FUNCTION_BLOCK FB_SXU
VAR_INPUT
	
END_VAR

VAR_OUTPUT
END_VAR



VAR
    // From lcls-srv01: grep -e KDes  /u1/lcls/epics/ioc/data/sioc-unds-uc*/iocInfo/IOC.pvlist |sort


    {attribute 'pytmc' := 'pv: 26; link: 2650:'}
    fbSegment_26 : FB_UndulatorSegment;
    
    {attribute 'pytmc' := 'pv: 27; link: 2750:'}
    fbSegment_27 : FB_UndulatorSegment;
    
    {attribute 'pytmc' := 'pv: 28; link: 2850:'}
    fbSegment_28 : FB_UndulatorSegment;
    
    {attribute 'pytmc' := 'pv: 29; link: 2950:'}
    fbSegment_29 : FB_UndulatorSegment;
    
    {attribute 'pytmc' := 'pv: 30; link: 3050:'}
    fbSegment_30 : FB_UndulatorSegment;
    
    {attribute 'pytmc' := 'pv: 31; link: 3150:'}
    fbSegment_31 : FB_UndulatorSegment;
    
    {attribute 'pytmc' := 'pv: 32; link: 3250:'}
    fbSegment_32 : FB_UndulatorSegment;
    
    {attribute 'pytmc' := 'pv: 33; link: 3350:'}
    fbSegment_33 : FB_UndulatorSegment;
    
    {attribute 'pytmc' := 'pv: 34; link: 3450:'}
    fbSegment_34 : FB_UndulatorSegment;
    
    {attribute 'pytmc' := 'pv: 36; link: 3650:'}
    fbSegment_36 : FB_UndulatorSegment;
    
    {attribute 'pytmc' := 'pv: 37; link: 3750:'}
    fbSegment_37 : FB_UndulatorSegment;
    
    {attribute 'pytmc' := 'pv: 38; link: 3850:'}
    fbSegment_38 : FB_UndulatorSegment;
    
    {attribute 'pytmc' := 'pv: 39; link: 3950:'}
    fbSegment_39 : FB_UndulatorSegment;
    
    {attribute 'pytmc' := 'pv: 40; link: 4050:'}
    fbSegment_40 : FB_UndulatorSegment;
    
    {attribute 'pytmc' := 'pv: 41; link: 4150:'}
    fbSegment_41 : FB_UndulatorSegment;
    
    {attribute 'pytmc' := 'pv: 42; link: 4250:'}
    fbSegment_42 : FB_UndulatorSegment;
    
    {attribute 'pytmc' := 'pv: 43; link: 4350:'}
    fbSegment_43 : FB_UndulatorSegment;
    
    {attribute 'pytmc' := 'pv: 44; link: 4450:'}
    fbSegment_44 : FB_UndulatorSegment;
    
    {attribute 'pytmc' := 'pv: 45; link: 4550:'}
    fbSegment_45 : FB_UndulatorSegment;
    
    {attribute 'pytmc' := 'pv: 46; link: 4650:'}
    fbSegment_46 : FB_UndulatorSegment;
    
    {attribute 'pytmc' := 'pv: 47; link: 4750:'}
    fbSegment_47 : FB_UndulatorSegment;
    


    fbSegment : ARRAY [iLowBound..iHighBound] OF POINTER TO FB_UndulatorSegment;
    fbCurrentSegment : REFERENCE TO FB_UndulatorSegment;

    iIndex : UDINT;

    bInitialized : BOOL := FALSE;

END_VAR

VAR CONSTANT
    iLowBound  : UDINT := 26;
    iHighBound : UDINT := 47;
END_VAR



IF NOT bInitialized THEN

    fbSegment[26] := ADR(fbSegment_26);
    fbSegment[27] := ADR(fbSegment_27);
    fbSegment[28] := ADR(fbSegment_28);
    fbSegment[29] := ADR(fbSegment_29);
    fbSegment[30] := ADR(fbSegment_30);
    fbSegment[31] := ADR(fbSegment_31);
    fbSegment[32] := ADR(fbSegment_32);
    fbSegment[33] := ADR(fbSegment_33);
    fbSegment[34] := ADR(fbSegment_34);
    fbSegment[35] := 0;
    fbSegment[36] := ADR(fbSegment_36);
    fbSegment[37] := ADR(fbSegment_37);
    fbSegment[38] := ADR(fbSegment_38);
    fbSegment[39] := ADR(fbSegment_39);
    fbSegment[40] := ADR(fbSegment_40);
    fbSegment[41] := ADR(fbSegment_41);
    fbSegment[42] := ADR(fbSegment_42);
    fbSegment[43] := ADR(fbSegment_43);
    fbSegment[44] := ADR(fbSegment_44);
    fbSegment[45] := ADR(fbSegment_45);
    fbSegment[46] := ADR(fbSegment_46);
    fbSegment[47] := ADR(fbSegment_47);

    bInitialized := TRUE;
END_IF

FOR iIndex := iLowBound TO iHighBound DO
    IF fbSegment[iIndex] <> 0 THEN
		fbCurrentSegment REF= fbSegment[iIndex]^;
		fbCurrentSegment();
    END_IF
END_FOR

END_FUNCTION_BLOCK

(* stored: Version 1.1.0.1, ProductVersion 3.1.4022.18
   POU FB_SXU: Id {23188e56-6a28-4c8b-9089-611f5a306284}, SpecialFunc None *)
